# EPICS alarm handler configuration: css_share/detectors/SVT/alh/SVT.R2.alhConfig
GROUP NULL R2
INCLUDE R2 SVT.R2.S1.alhConfig
INCLUDE R2 SVT.R2.S2.alhConfig
INCLUDE R2 SVT.R2.S3.alhConfig
INCLUDE R2 SVT.R2.S4.alhConfig
INCLUDE R2 SVT.R2.S5.alhConfig
INCLUDE R2 SVT.R2.S6.alhConfig
INCLUDE R2 SVT.R2.S7.alhConfig
INCLUDE R2 SVT.R2.S8.alhConfig
INCLUDE R2 SVT.R2.S9.alhConfig
INCLUDE R2 SVT.R2.S10.alhConfig
INCLUDE R2 SVT.R2.S11.alhConfig
INCLUDE R2 SVT.R2.S12.alhConfig
INCLUDE R2 SVT.R2.S13.alhConfig
INCLUDE R2 SVT.R2.S14.alhConfig
